TYPE "Decoiler_Manager"
VERSION : 0.1
// Block: Decoiler_Manager
   STRUCT
      IsOutLine : Bool;
      IsInLine : Bool;
      EmptiyngConfirmed : Bool;
      ModePneumaticBraking : Bool;
      TotalBrakeOpeningAttempt : Bool;
      Feed : SpeedMachine_CIn_Manager;
      Coupling : ValveMachine_Manager;
      Jaws : ValveMachine_Manager;
      SnubberLift : ValveMachine_Manager;
      SnubberRoll : ValveMachine_Manager;
   END_STRUCT;

END_TYPE
